FUNCTION_BLOCK F_CTRL_IN (* Basic Function Block Type *)
  (* Standard: 61499-2; Classification: control module; Description: CTRL_IN calculates the process deviation (SET_POINT _ ACTUAL) and passes them at the output. If the diference is less than the value at the input  NOISE of the output remains at 0. CTRL_IN can be used to build own rule modules. *)
  (* Version 0.0, 2011-08-23, 4DIAC-IDE, 4DIAC-Consortium *)
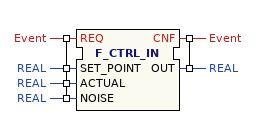
  EVENT_INPUT
    REQ WITH ACTUAL, NOISE, SET_POINT; (* Normal Execution Request *)
  END_EVENT
  EVENT_OUTPUT
    CNF WITH OUT; (* Execution Confirmation *)
  END_EVENT
  VAR_INPUT
    SET_POINT : REAL; (* default *)
    ACTUAL : REAL; (* process value *)
    NOISE : REAL; (* threshold *)
  END_VAR
  VAR_OUTPUT
    OUT : REAL; (* process deviation *)
  END_VAR
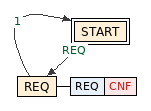
  EC_STATES
    START; (* Initial State *)
    REQ : REQ -> CNF; (* Normal execution *)
  END_STATES
  EC_TRANSITIONS
    START TO REQ := REQ;
    REQ TO START := 1;
  END_TRANSITIONS
  ALGORITHM REQ IN ST: (* Normally executed algorithm *)
CTRL_IN := DEAD_ZONE(SET_POINT - ACTUAL, NOISE);
  END_ALGORITHM
END_FUNCTION_BLOCK
